//{{V2}}
FUNCTION_BLOCK FB1
TITLE=   <Title of FB>


AUTHOR:nb
FAMILY:nb
NAME:nb
VERSION:1.0


VAR_INPUT
END_VAR

VAR_OUTPUT
END_VAR

VAR_IN_OUT
END_VAR

VAR
END_VAR

VAR_TEMP
END_VAR
BEGIN

NETWORK
TITLE=   <Title of Network>
//{{a}}




END_FUNCTION_BLOCK
